FUNCTION_BLOCK Q_ObjEnableDisable (* Command enable/disable (input) object - ( Part 6 - F.4 ) *)
  (* Standard: ISO 11783-6; Description: This command is used to enable or disable an input field object and pertains to the accessibility of an input object. Return values iso_s16 - E_NO_ERR - OK - E_OVERFLOW - buffer overflow - E_NOACT - Command not possible in current state - E_NO_INSTANCE - No VT client available *)
  (* Version 1.0, 2022-07-08, franz *)
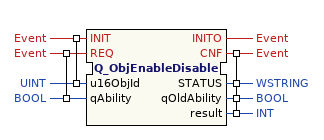
  EVENT_INPUT
    INIT WITH u16ObjId; (* Service Initialization *)
    REQ WITH qAbility; (* Service Request *)
  END_EVENT
  EVENT_OUTPUT
    INITO; (* Initialization Confirm *)
    CNF WITH STATUS, qOldAbility, result; (* Confirmation of Requested Service *)
  END_EVENT
  VAR_INPUT
    u16ObjId : UINT; (* Object ID *)
    qAbility : BOOL; (* 0 == disable, 1 == enable *)
  END_VAR
  VAR_OUTPUT
    STATUS : WSTRING; (* Service Status *)
    qOldAbility : BOOL; (* 0 == disable, 1 == enable *)
    result : INT; (* retval see description *)
  END_VAR
END_FUNCTION_BLOCK
